Fanuc KAREL source: SET_FILE_POS.kl

PROGRAM T
%NOLOCKGROUP
VAR
 v0 : FILE
 v1 : INTEGER
 v2 : INTEGER
BEGIN
 SET_FILE_POS(v0, v1, v2)
END T
